// TIA Portal V21 export
FUNCTION "Main dispositivi profinet" : Void   // FC98, LAD
{ S7_Optimized_Access := 'TRUE' }
// stored: SetENOAutomatically false
BEGIN

REGION Network 1 (SCL)
   "GestProfinetDiagnostica"();
   "GestProfinetAbilitazionedispositivo"();
END_REGION
END_FUNCTION
